FUNCTION_BLOCK EP7402CH1
VAR_INPUT
END_VAR
VAR_OUTPUT
END_VAR
VAR
	EP7402DigIn1 AT%I* : BOOL;
	EP7402ReadyToEnable AT%I* : BOOL;
	EP7402Ready AT%I* : BOOL;
	EP7402Warning AT%I* : BOOL;
	EP7402Error AT%I* : BOOL;
	EP7402MovingPos AT%I* : BOOL;
	EP7402MovingNeg AT%i* : BOOL;
	EP7402Enable AT%Q* : BOOL;
	EP7402InvertDirection AT%Q* : BOOL;
	EP7402Velocity AT%q* : INT;
END_VAR

METHOD Disable : BOOL
VAR_INPUT
END_VAR
EP7402Enable := false;
END_METHOD

METHOD Enable : BOOL
VAR_INPUT
END_VAR
EP7402Enable := TRUE;
END_METHOD

METHOD MoveNeg : BOOL
VAR_INPUT
END_VAR
EP7402InvertDirection := TRUE;
	EP7402Velocity := 6000;
END_METHOD

METHOD MovePos : BOOL
VAR_INPUT
END_VAR
EP7402Velocity := 6000;
END_METHOD

METHOD Stop : BOOL
VAR_INPUT
END_VAR
EP7402Velocity := 0;
END_METHOD

END_FUNCTION_BLOCK

(* stored: Version 1.1.0.1, ProductVersion 3.1.4024.9
   POU EP7402CH1: Id {6c5f7c1d-1191-4da5-ba6c-9233e15b621c}, SpecialFunc None
   Method Disable: Id {a3bf5df0-9c23-4707-adfd-85b9fcedd433}
   Method Enable: Id {69b44551-5844-42d2-b1fb-69cd7479da38}
   Method MoveNeg: Id {b2140de2-50ba-45d3-8d0c-e25d3c8c6c62}
   Method MovePos: Id {cfec3af2-c578-4937-a526-cc8a734135af}
   Method Stop: Id {cf5a21b5-0585-43bb-ad8d-f1808560a28e} *)
